(* IEC 61131-3 sources: eCockpitGit/test_project/src/%F%00 Library/%F%Common Functions/%F%String/%F%Address Input/%F%Len, 2 files *)

(* ---- %POU%FU_LenAI.st ---- *)
//This function, returns the lenght of a string of any size from a pointer
//Input string must be zero terminated
// |**Version**|**Author**| **Date** |**Changes**
// | 1         | NSN      | 16-09-20 | Creation
FUNCTION FU_LenAI : DWORD
VAR_INPUT
	str			:POINTER TO EASCII;			//Input String
END_VAR
(*%!%__DELIMITER__%!%*)
IF str <> 0 THEN
	WHILE str^ <> 0 DO
		FU_LenAI		:=		FU_LenAI + 1;
		str				:=		str + 1;
	END_WHILE
END_IF

(* ---- %POU%FU_wLenAI.st ---- *)
//This function, returns the lenght of a string of any size from a pointer
//Input string must be zero terminated
// |**Version**|**Author**| **Date** |**Changes**
// | 1         | NSN      | 16-09-20 | Creation
FUNCTION FU_wLenAI : WORD
VAR_INPUT
	str			:POINTER TO EASCII;			//Input String
END_VAR
(*%!%__DELIMITER__%!%*)
IF str <> 0 THEN
	WHILE str^ <> 0 DO
		FU_wLenAI		:=		FU_wLenAI + 1;
		str				:=		str + 1;
	END_WHILE
END_IF
